(* PLC project FB_OUTPUT_DIMMER_DALI_MQTT, WAGO e!COCKPIT e!COCKPIT *)
(* stored: creationDateTime 2026-02-03T13:38:40.6404858, modificationDateTime 2026-02-03T13:38:16.7598415 *)

{attribute 'reflection'}
FUNCTION_BLOCK FB_OUTPUT_DIMMER_DALI_MQTT EXTENDS FB_MQTT_BASE IMPLEMENTS MQTT.MQTT_SUBSCRIBE_CALLBACK
  VAR_INPUT
    BALLAST : typBallast;
    TOGGLE : BOOL;
    P_LONG : BOOL;
    PRIO_HIGH : BOOL := FALSE;
    PRIO_LOW : BOOL := FALSE;
  END_VAR
  VAR_OUTPUT
    STATUS_LED : BOOL;
  END_VAR
  VAR
    {attribute 'instance-path'}
    {attribute 'noinit'}
    InstancePath : STRING;  (* Refelection: object's full instance name *)
    Startup : BOOL := TRUE;
    DaliSendDimValue : FbDaliSendDimValue;
    DaliSendFadeTime : FbDaliSendFadeTime;
    DaliSendFadeRate : FbDaliSendFadeRate;
    MqttSendBrightnessUpdate : BOOL;
    MqttSendOnUpdate : BOOL;
    MqttSendOffUpdate : BOOL;
    Toggle_RTrigger : Standard.R_TRIG;
    DaliSyncSignalGenerator : Util.BLINK;
    DaliConfigSyncSignalGenerator : Util.BLINK;
    DimDirection : INT := 1;
  END_VAR
  VAR PERSISTENT
    DimValue : REAL;
  END_VAR

            DaliSendFadeTime(
	typBallast := BALLAST,
	bFadeTime := 2, // 1 sec
	xUpdate := DaliConfigSyncSignalGenerator.OUT
	);
	
DaliSendFadeRate(
	typBallast := BALLAST,
	bFadeRate := 2, // 1 sec
	xUpdate := DaliConfigSyncSignalGenerator.OUT
	);

DaliSendDimValue(
	typBallast := BALLAST,
	rDimValue := DimValue,
	xUpdate := DaliSyncSignalGenerator.OUT OR MqttSendOffUpdate OR MqttSendOnUpdate);

DaliSyncSignalGenerator(
	ENABLE := TRUE,
	TIMEHIGH := T#1S,
	TIMELOW := T#1M);
	
DaliConfigSyncSignalGenerator(
	ENABLE := TRUE,
	TIMEHIGH := T#1S,
	TIMELOW := T#24H);

Toggle_RTrigger(CLK:=TOGGLE);

// Regular push
IF(Toggle_RTrigger.Q AND DimValue = 0) THEN
	SetDimValue(100);
ELSIF(Toggle_RTrigger.Q AND DimValue > 0) THEN
	SetDimValue(0);
END_IF

// Long push
IF P_LONG THEN
	SetDimValue(DimValue + DimDirection);
END_IF

IF MqttSendBrightnessUpdate OR Startup AND InitMqttDone THEN
	pMqttPublishQueue^.AddMessage(		
		Payload := REAL_TO_STRING(DimValue),
		Topic := CONCAT(THIS^.MQTTPublishTopic, '/BRIGHTNESS'),
		Qos := MQTT.QoS.ExactlyOnce,
		MqttRetain := TRUE
	);
	MqttSendBrightnessUpdate := FALSE;
END_IF

IF MqttSendOnUpdate OR (Startup AND DimValue > 0) AND InitMqttDone THEN
	pMqttPublishQueue^.AddMessage(		
		Payload := 'ON',
		Topic := THIS^.MQTTPublishTopic,
		Qos := MQTT.QoS.ExactlyOnce,
		MqttRetain := TRUE
	);
	MqttSendOnUpdate := FALSE;
END_IF

IF MqttSendOffUpdate OR (Startup AND DimValue = 0) AND InitMqttDone THEN
	pMqttPublishQueue^.AddMessage(
		Payload := 'OFF',
		Topic := THIS^.MQTTPublishTopic,
		Qos := MQTT.QoS.ExactlyOnce,
		MqttRetain := TRUE
	);
	MqttSendOffUpdate := FALSE;
END_IF

Startup:=FALSE;
STATUS_LED := REAL_TO_BOOL(DimValue);
          

METHOD InitMqttDiscovery
  VAR_INPUT
    Device : POINTER TO FB_PLC_MQTT_DISCOVERY_DEVICE;
    Name : STRING(255);
    overruleId : STRING(255) := '';
    meta : STRING(255) := '';
  END_VAR
  VAR
    id : STRING(255);
  END_VAR
                  IF InitMqttDone AND NOT initMqttDiscoveryDone THEN
	
	IF CommonTypesAndFunctions.StrEquals(str1:= ADR(overruleId), str2:= ADR('')) THEN
		id := CONCAT(CONCAT(THIS^.DeviceName,'_'), THIS^.InstanceNamePt^); // 'FB_DI_PB_003'
	ELSE
		id := overruleId; // 'MY_PH_GND_HALL_01'
	END_IF
	
	Device^.CreateLightDimmerEntity(
		Name := name,
		Id := Id,
		Meta := meta,
		CommandTopic := THIS^.MQTTSubscribeTopic,
		PayloadOn := 'ON',
		PayloadOff := 'OFF',
		StateTopic := THIS^.MQTTPublishTopic,
		BrightnessCommandTopic := CONCAT(THIS^.MQTTSubscribeTopic, '/BRIGHTNESS'),
		BrightnessStateTopic := CONCAT(THIS^.MQTTPublishTopic, '/BRIGHTNESS'),
		BrightnessScale := 100,
		OnCommandType := 'brightness');

	initMqttDiscoveryDone := TRUE;
END_IF
                
END_METHOD

METHOD InitMqtt
  VAR_INPUT
    MQTTPublishPrefix : POINTER TO STRING;
    MQTTSubscribePrefix : POINTER TO STRING;
    pMqttPublishQueue : POINTER TO FB_MqttPublishQueue;
    pMqttCallbackCollector : POINTER TO MQTT.CallbackCollector;
  END_VAR
                  SUPER^._InstancePath := THIS^.InstancePath; // Due to reflection its location is important

(*pass trough*)
THIS^.pMqttPublishQueue := pMqttPublishQueue;
THIS^.MqttPublishTopicPrefix:=MQTTPublishPrefix;
THIS^.MQTTSubscribeTopicPrefix:=MQTTSubscribePrefix;
THIS^.pMqttPublishQueue:=pMqttPublishQueue;

SUPER^.InitBaseMqtt();
pMqttCallbackCollector^.put(instance:= THIS^); // register the FB agains the collector so mqtt events can be received


                
END_METHOD

METHOD PublishReceived : BOOL
  VAR_INPUT
    Data : MQTT.CALLBACK_DATA;  (* Collection of recived Data *)
  END_VAR
                  //first check if Mqtt is initialized, otherwise do nothing
IF NOT(InitMqttDone) THEN
	//mark the interface call from the collector as done
	PublishReceived := TRUE;
	
ELSIF MQTTSubscribeTopic =  Data.TopicOut^ THEN
	IF CommonTypesAndFunctions.StrEquals(str1:= Data.PayloadString, str2:= ADR('ON')) THEN
		SetDimValue(100);
	ELSIF CommonTypesAndFunctions.StrEquals(str1:= Data.PayloadString, str2:= ADR('OFF')) THEN
		SetDimValue(0);
	END_IF
	
ELSIF CONCAT(MQTTSubscribeTopic, '/BRIGHTNESS') =  Data.TopicOut^ THEN
	IF OSCAT_BASIC.IS_CC(str:= Data.PayloadString^,cmp:='0123456789.') AND THIS^.PRIO_HIGH = FALSE THEN
		SetDimValue(STRING_TO_REAL(Data.PayloadString^));
	END_IF
END_IF 
                
END_METHOD

METHOD SetDimValue
  VAR_INPUT
    Value : REAL;
  END_VAR
                  THIS^.MqttSendBrightnessUpdate := TRUE;

IF THIS^.DimValue = 0 AND Value > 0 THEN
	THIS^.MqttSendOnUpdate := TRUE;
END_IF

IF THIS^.DimValue > 0 AND Value = 0 THEN
	THIS^.MqttSendOffUpdate := TRUE;
END_IF

IF Value = 0 THEN
	DimDirection := 1;
ELSIF Value = 100 THEN
	DimDirection := -1;
END_IF

THIS^.DimValue := Value;
                
END_METHOD

METHOD ConfigureFunctionBlock : BOOL
  VAR_INPUT
    FadeTime : BYTE;
    FadeRate : BYTE;
  END_VAR
                  DaliSendFadeTime.bFadeTime := FadeTime;
DaliSendFadeRate.bFadeRate := FadeRate;
                
END_METHOD
END_FUNCTION_BLOCK
